// Created by Dimitar Stojanov 06.2023 
// Install TC2_Utilities and Import ST_Time structure for fully functionality of this block


FUNCTION_BLOCK FB_SystemDateTime
VAR_INPUT
	CustomBlink1_ON		:TIME;
	CustomBlink1_OFF	:TIME;
	CustomBlink2_ON		:TIME;
	CustomBlink2_OFF	:TIME;
	CustomBlink3_ON		:TIME;
	CustomBlink3_OFF	:TIME;
END_VAR
VAR_OUTPUT
	dtDateTime		:DT;
	sTime			:STRING;
	sDate			:STRING;
	sDateTime		:STRING;
	sFormatDateTime	:STRING;
	Clock_500ms		:BOOL;
	Clock_1s		:BOOL;
	Clock_2s		:BOOL;
	Clock_5s		:BOOL;
	Clock_60s		:BOOL;
	Clock_1sOFF_2sON	:BOOL;
	Pulse_10s		:BOOL;
	Pulse_30s		:BOOL;
	Pulse_60s		:BOOL;
	CustomBlink1	:BOOL;
	CustomBlink2	:BOOL;
	CustonBlink3	:BOOL;
	newHour			:BOOL; //true for 1 cycle when hour change
	newDay			:BOOL;
	newMonth		:BOOL;
	newYear			:BOOL;
END_VAR
VAR
	bFirstCycle		:BOOL:=TRUE;	

	fbTime			:FB_LocalSystemTime;
	systemDateTime	:TIMESTRUCT;
	
	Second			:STRING;
	Minute			:STRING;
	Hour			:STRING;
	Day				:STRING;
	Month			:STRING;
	Year			:STRING;
	
	iClock1s		:INT;
	TON_0: TON;
	TOF_0: TOF;
	TON_1: TON;
	TOF_1: TOF;
	TOF_2: TOF;
	TON_2: TON;
	TON_3: TON;
	TOF_3: TOF;
	TOF_4: TOF;
	TON_4: TON;
	TON_5: TON;
	TOF_5: TOF;
	TON_6: TON;
	TOF_6: TOF;
	TON_7: TON;
	TOF_7: TOF;
	TON_8: TON;
	TOF_8: TOF;
	
	TON_9: TON;
	TOF_9: TOF;
	TOF_10: TOF;
	TOF_11: TOF;
	TON_10: TON;
	TON_20: TON;
	TOF_20: TOF;
	TON_21: TON;
	TOF_21: TOF;
	TON_22: TON;
	TOF_22: TOF;
	
	TOF_23: TOF;
	
	bDelay			:BOOL;
	TON_DELAY		:TON;
END_VAR

VAR_OUTPUT PERSISTENT
	CurrentHour		:WORD;
	CurrentDay		:WORD;
	CurrentMonth	:WORD;
	CurrentYear		:WORD;
END_VAR

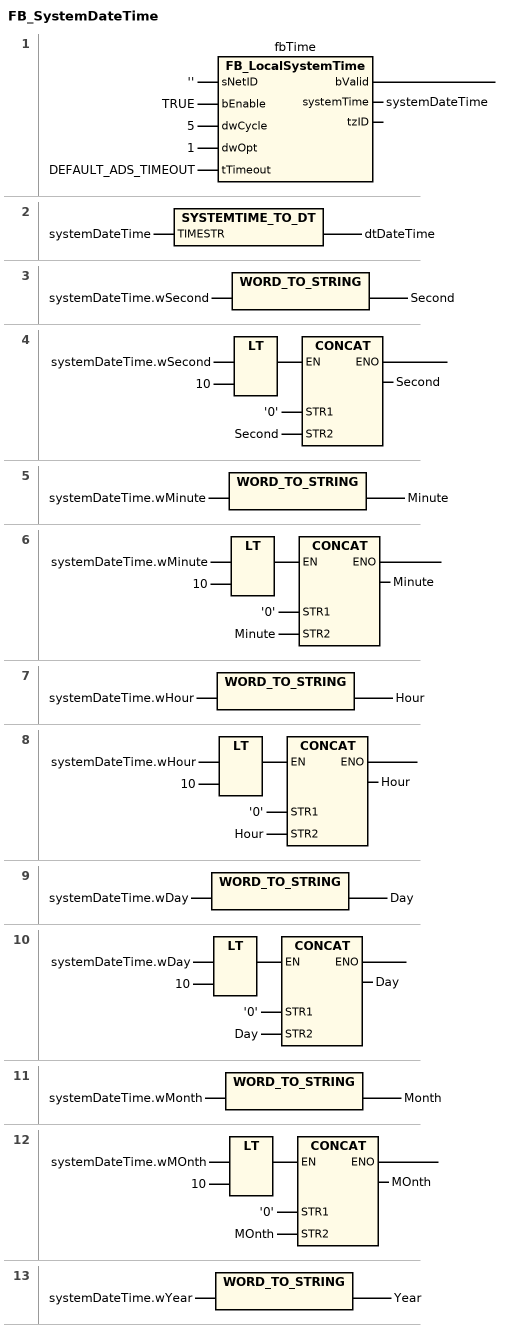
// NETWORK 1
fbTime(
    sNetID := '',
    bEnable := TRUE,
    dwCycle := 5,
    dwOpt := 1,
    tTimeout := DEFAULT_ADS_TIMEOUT,
    systemTime => systemDateTime); // FB_LocalSystemTime

// NETWORK 2
dtDateTime := SYSTEMTIME_TO_DT(TIMESTR := systemDateTime);

// NETWORK 3
Second := WORD_TO_STRING(systemDateTime.wSecond);

// NETWORK 4
IF systemDateTime.wSecond < 10 THEN Second := CONCAT(STR1 := '0', STR2 := Second); END_IF

// NETWORK 5
Minute := WORD_TO_STRING(systemDateTime.wMinute);

// NETWORK 6
IF systemDateTime.wMinute < 10 THEN Minute := CONCAT(STR1 := '0', STR2 := Minute); END_IF

// NETWORK 7
Hour := WORD_TO_STRING(systemDateTime.wHour);

// NETWORK 8
IF systemDateTime.wHour < 10 THEN Hour := CONCAT(STR1 := '0', STR2 := Hour); END_IF

// NETWORK 9
Day := WORD_TO_STRING(systemDateTime.wDay);

// NETWORK 10
IF systemDateTime.wDay < 10 THEN Day := CONCAT(STR1 := '0', STR2 := Day); END_IF

// NETWORK 11
Month := WORD_TO_STRING(systemDateTime.wMonth);

// NETWORK 12
IF systemDateTime.wMOnth < 10 THEN MOnth := CONCAT(STR1 := '0', STR2 := MOnth); END_IF

// NETWORK 13
Year := WORD_TO_STRING(systemDateTime.wYear);

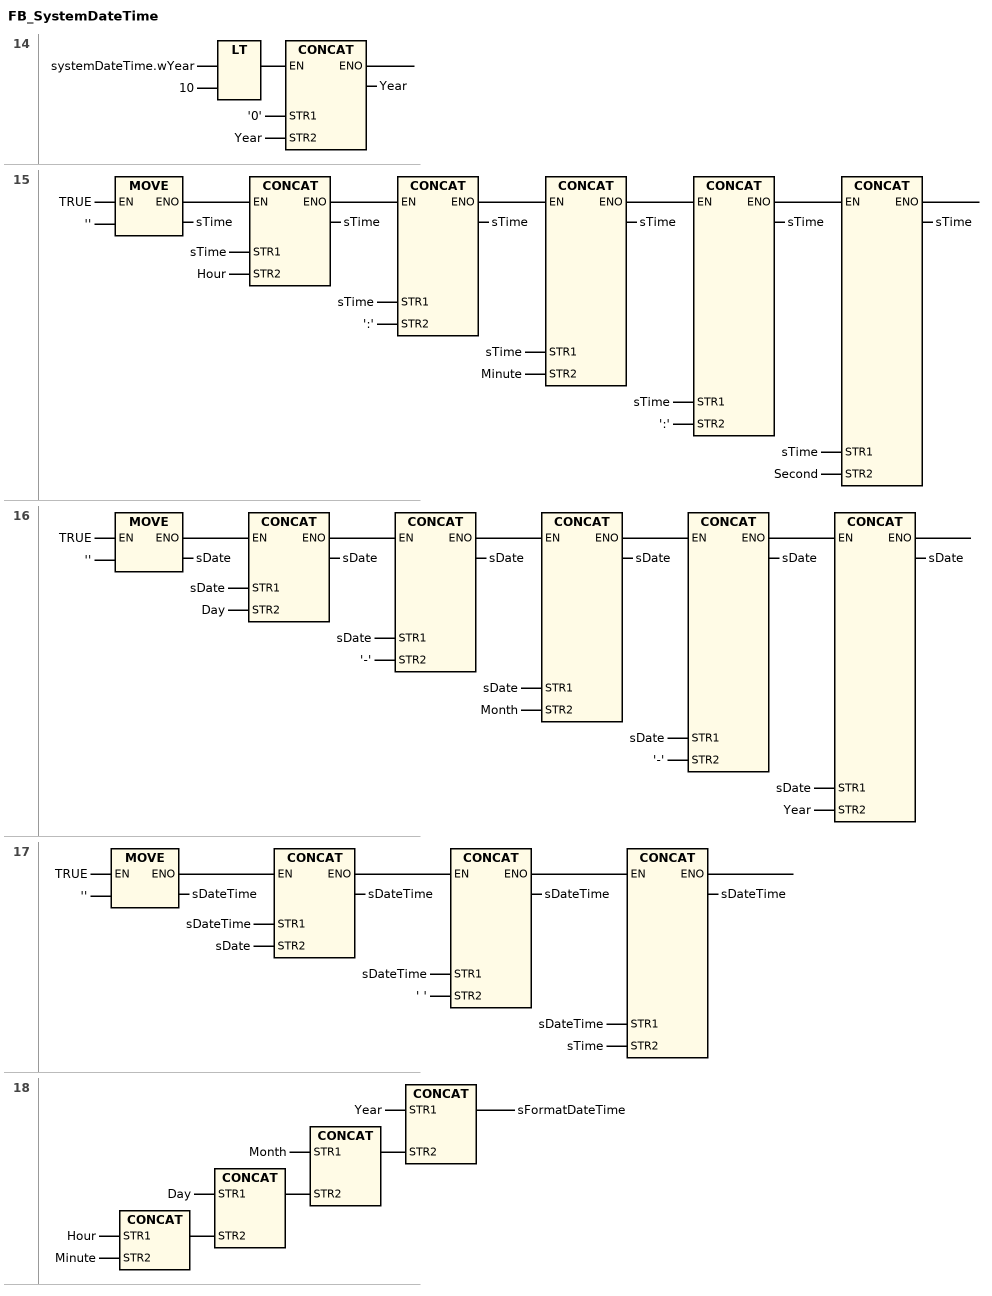
// NETWORK 14
IF systemDateTime.wYear < 10 THEN Year := CONCAT(STR1 := '0', STR2 := Year); END_IF

// NETWORK 15
sTime := '';
sTime := CONCAT(STR1 := sTime, STR2 := Hour);
sTime := CONCAT(STR1 := sTime, STR2 := ':');
sTime := CONCAT(STR1 := sTime, STR2 := Minute);
sTime := CONCAT(STR1 := sTime, STR2 := ':');
sTime := CONCAT(STR1 := sTime, STR2 := Second);

// NETWORK 16
sDate := '';
sDate := CONCAT(STR1 := sDate, STR2 := Day);
sDate := CONCAT(STR1 := sDate, STR2 := '-');
sDate := CONCAT(STR1 := sDate, STR2 := Month);
sDate := CONCAT(STR1 := sDate, STR2 := '-');
sDate := CONCAT(STR1 := sDate, STR2 := Year);

// NETWORK 17
sDateTime := '';
sDateTime := CONCAT(STR1 := sDateTime, STR2 := sDate);
sDateTime := CONCAT(STR1 := sDateTime, STR2 := ' ');
sDateTime := CONCAT(STR1 := sDateTime, STR2 := sTime);

// NETWORK 18
sFormatDateTime := CONCAT(STR1 := Year, STR2 := CONCAT(STR1 := Month, STR2 := CONCAT(STR1 := Day, STR2 := CONCAT(STR1 := Hour, STR2 := Minute))));

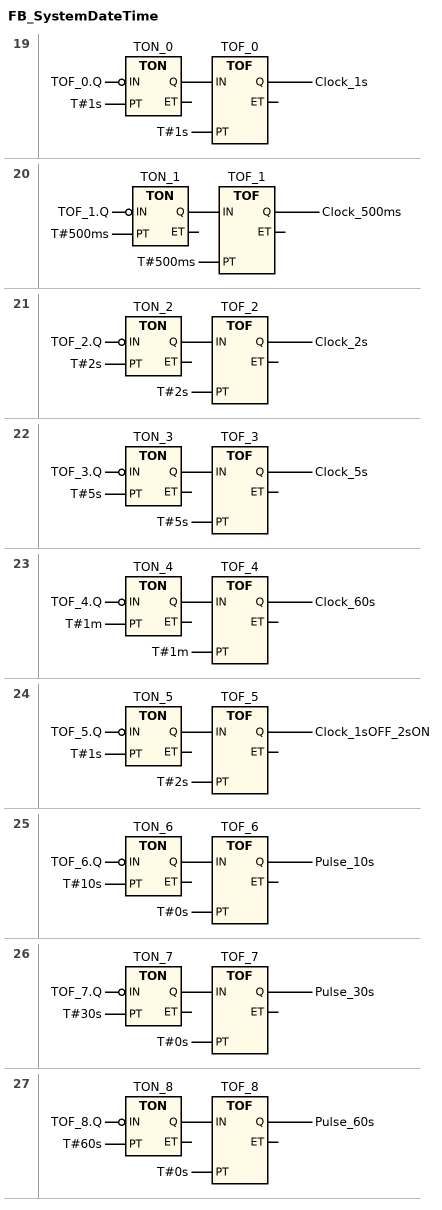
// NETWORK 19
TON_0(IN := NOT TOF_0.Q, PT := T#1s); // TON
TOF_0(IN := TON_0.Q, PT := T#1s); // TOF
Clock_1s := TOF_0.Q;

// NETWORK 20
TON_1(IN := NOT TOF_1.Q, PT := T#500ms); // TON
TOF_1(IN := TON_1.Q, PT := T#500ms); // TOF
Clock_500ms := TOF_1.Q;

// NETWORK 21
TON_2(IN := NOT TOF_2.Q, PT := T#2s); // TON
TOF_2(IN := TON_2.Q, PT := T#2s); // TOF
Clock_2s := TOF_2.Q;

// NETWORK 22
TON_3(IN := NOT TOF_3.Q, PT := T#5s); // TON
TOF_3(IN := TON_3.Q, PT := T#5s); // TOF
Clock_5s := TOF_3.Q;

// NETWORK 23
TON_4(IN := NOT TOF_4.Q, PT := T#1m); // TON
TOF_4(IN := TON_4.Q, PT := T#1m); // TOF
Clock_60s := TOF_4.Q;

// NETWORK 24
TON_5(IN := NOT TOF_5.Q, PT := T#1s); // TON
TOF_5(IN := TON_5.Q, PT := T#2s); // TOF
Clock_1sOFF_2sON := TOF_5.Q;

// NETWORK 25
TON_6(IN := NOT TOF_6.Q, PT := T#10s); // TON
TOF_6(IN := TON_6.Q, PT := T#0s); // TOF
Pulse_10s := TOF_6.Q;

// NETWORK 26
TON_7(IN := NOT TOF_7.Q, PT := T#30s); // TON
TOF_7(IN := TON_7.Q, PT := T#0s); // TOF
Pulse_30s := TOF_7.Q;

// NETWORK 27
TON_8(IN := NOT TOF_8.Q, PT := T#60s); // TON
TOF_8(IN := TON_8.Q, PT := T#0s); // TOF
Pulse_60s := TOF_8.Q;

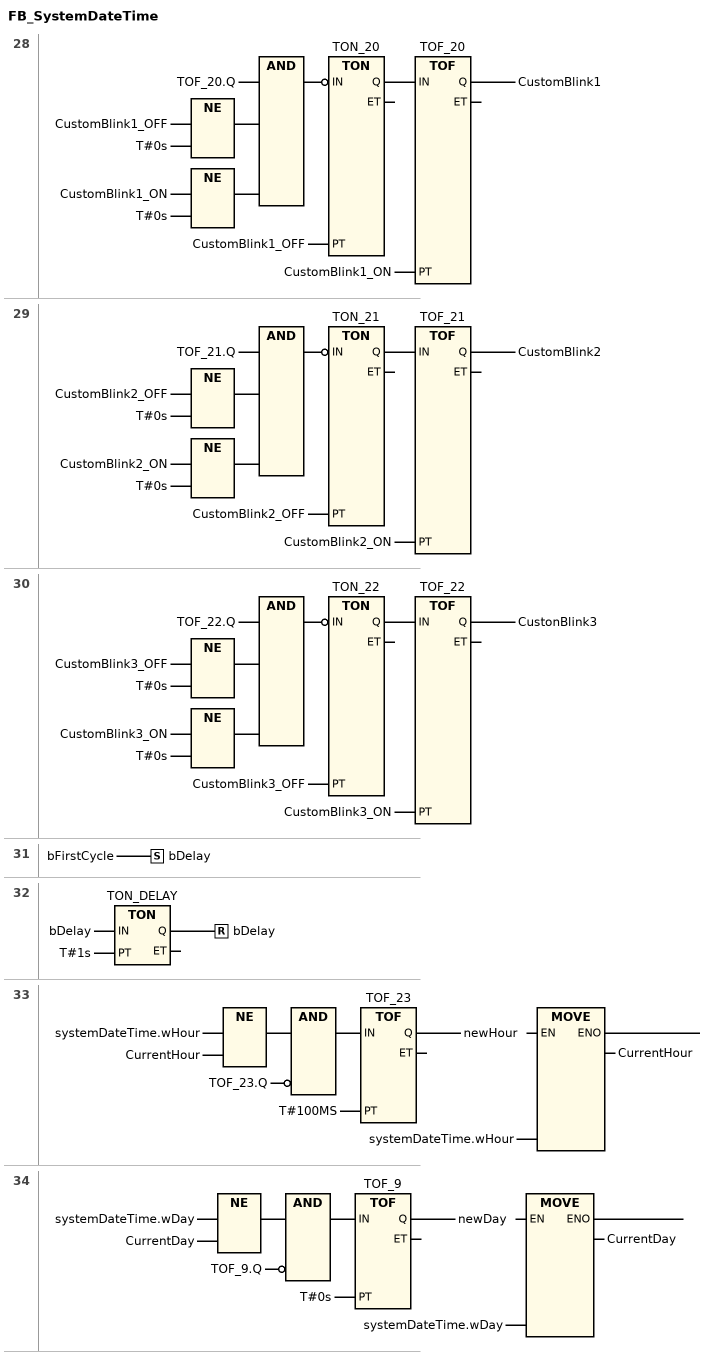
// NETWORK 28
TON_20(IN := NOT (TOF_20.Q AND CustomBlink1_OFF <> T#0s AND CustomBlink1_ON <> T#0s), PT := CustomBlink1_OFF); // TON
TOF_20(IN := TON_20.Q, PT := CustomBlink1_ON); // TOF
CustomBlink1 := TOF_20.Q;

// NETWORK 29
TON_21(IN := NOT (TOF_21.Q AND CustomBlink2_OFF <> T#0s AND CustomBlink2_ON <> T#0s), PT := CustomBlink2_OFF); // TON
TOF_21(IN := TON_21.Q, PT := CustomBlink2_ON); // TOF
CustomBlink2 := TOF_21.Q;

// NETWORK 30
TON_22(IN := NOT (TOF_22.Q AND CustomBlink3_OFF <> T#0s AND CustomBlink3_ON <> T#0s), PT := CustomBlink3_OFF); // TON
TOF_22(IN := TON_22.Q, PT := CustomBlink3_ON); // TOF
CustonBlink3 := TOF_22.Q;

// NETWORK 31
bDelay S= bFirstCycle;

// NETWORK 32
TON_DELAY(IN := bDelay, PT := T#1s); // TON
bDelay R= TON_DELAY.Q;

// NETWORK 33
TOF_23(IN := systemDateTime.wHour <> CurrentHour AND NOT TOF_23.Q, PT := T#100MS); // TOF
newHour := TOF_23.Q;
IF TOF_23.Q THEN CurrentHour := systemDateTime.wHour; END_IF

// NETWORK 34
TOF_9(IN := systemDateTime.wDay <> CurrentDay AND NOT TOF_9.Q, PT := T#0s); // TOF
newDay := TOF_9.Q;
IF TOF_9.Q THEN CurrentDay := systemDateTime.wDay; END_IF

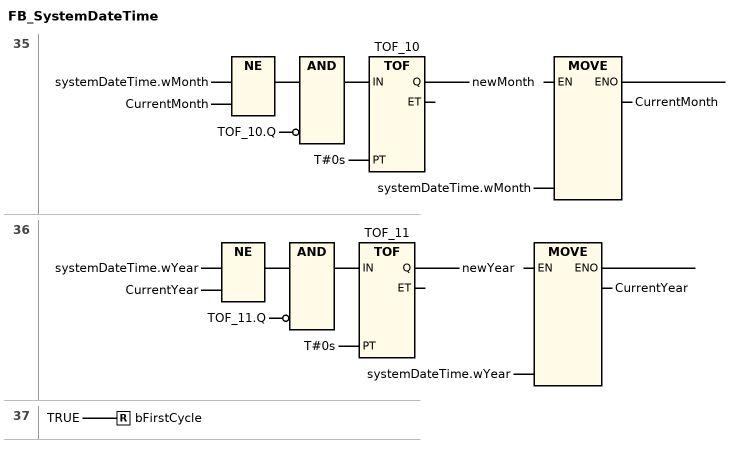
// NETWORK 35
TOF_10(IN := systemDateTime.wMonth <> CurrentMonth AND NOT TOF_10.Q, PT := T#0s); // TOF
newMonth := TOF_10.Q;
IF TOF_10.Q THEN CurrentMonth := systemDateTime.wMonth; END_IF

// NETWORK 36
TOF_11(IN := systemDateTime.wYear <> CurrentYear AND NOT TOF_11.Q, PT := T#0s); // TOF
newYear := TOF_11.Q;
IF TOF_11.Q THEN CurrentYear := systemDateTime.wYear; END_IF

// NETWORK 37
bFirstCycle R= TRUE;

END_FUNCTION_BLOCK

(* stored: Version 1.1.0.1
   POU FB_SystemDateTime: Id {96075684-39ec-474a-a046-d45c9c1209eb}, SpecialFunc None *)
